Omron Sysmac Studio project ReplaceStrFB (Sysmac Studio 1.62.0.64009, StandardProject)

# Controller new_Controller_0: NX102-9000 version 1.68
Task PrimaryTask (priority 4, period or condition 2000): Sample

PROGRAM Sample
VAR
    test : BOOL;
    InStr : STRING[1986];
    OldStr : STRING[256];
    NewStr : STRING[256];
    OutStr : STRING[1986];
    Replaced : BOOL;
END_VAR
VAR
    _e1 : R_TRIG;
    _e2 : R_TRIG;
END_VAR

(* Section Section0: ladder, written here as Structured Text *)

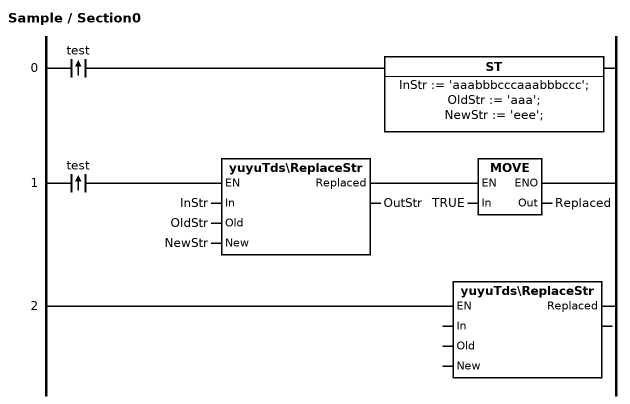
(* Rung 0 *)
_e1(CLK := test);
IF _e1.Q THEN
    InStr := 'aaabbbcccaaabbbccc';
    OldStr := 'aaa';
    NewStr := 'eee';
END_IF;
(* Rung 1 *)
_e2(CLK := test);
IF _e2.Q THEN OutStr := yuyuTds\ReplaceStr(In := InStr, Old := OldStr, New := NewStr); END_IF;
IF OutStr THEN Replaced := TRUE; END_IF;
(* Rung 2 *)
END_PROGRAM

FUNCTION yuyuTds\ReplaceStr : STRING[1986]  (* 置換後の文字列 *)
VAR
    Pos : UINT;
END_VAR
VAR_INPUT
    In : STRING[1986];  (* 元の文字列 *)
    Old : STRING[256];  (* 検索する文字列 *)
    New : STRING[256];  (* 置き換える文字列 *)
END_VAR
VAR_OUTPUT
    Replaced : BOOL;  (* 置換有無結果 (TRUE:置換有 FALSE:置換無) *)
END_VAR
Pos := FIND(In1:=In, In2:=Old);

IF Pos = 0 THEN
	// 検索文字がない場合（置換しない場合）
	ReplaceStr := In;
	Replaced := FALSE;
ELSE
	// 検索文字がある場合（置換する場合）
	ReplaceStr := REPLACE(In1:=In, In2:=New, L:=LEN(Old), P:=Pos);
	Replaced := TRUE;
END_IF;
END_FUNCTION